# EPICS autosave request: trunk/stdApp/Db/femto_DHPCA_100.req
$(P)$(A):Description
$(P)$(A):GainIndex
$(P)$(A):Coupling
$(P)$(A):Filter
